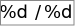
VISUALIZATION VI_NumberHollow  // 75x26
VAR_IN_OUT
	nNumberToDisplay : INT;
	nMaxNumberToDisplay : INT;
END_VAR
    Rectangle (-3,0 34x24), "%d", text variable: nNumberToDisplay
    Rectangle (41,0 32x24), "%d", text variable: nMaxNumberToDisplay
    Rectangle (27,0 17x24), "/", text variable: GVL_XtsVisuLib.nXtsIdMaxToDisplay
END_VISUALIZATION

(* stored: Version 1.1.0.1, ProductVersion 3.1.4024.9
   Visu VI_NumberHollow: Id {fb97838e-2148-4bc3-ac2f-a168376a8c1d} *)
